FUNCTION_BLOCK FB_ErrorList

VAR_INPUT
	En : BOOL;											//Enable input
	bReset : BOOL;										//Delete all Error entry
	lErrorID : ULINT;									//ErrorID to be acknoledged
	bACK : BOOL;										//Acknoledge the given error and delete it from the list
END_VAR
	
VAR_OUTPUT
	EnO : BOOL;											//Enable output
	nNoError: UINT;										//Number of Errors
	nNoOverflow : INT;									//Number of Overflows
	pErrorSystem : POINTER TO ST_ErrorSystem;			//Pointer to ErrorSystem
END_VAR

VAR
	nFreePos : UINT;									//Number of free position in the list
	nListCnt1 : UINT;									//work variable
	ErrorSystem : ST_ErrorSystem;						//Data structure of the Error list
END_VAR

(*
* ================================================================================
*                                   DESCRIPTION
* ================================================================================
* This Function Block implements the core structure of the Error/Warning Handling
* system. It realizes the datastructure containing every Error Entry, collect
* statistics about the usage and manage the Error Entries.
* Note: The system is under development, most of the functionalities are not
* implemented or existing functionalities may change with the advance of the
* development.
* ================================================================================
*)
EnO := En;

//Ponter to ErrorSystem
pErrorSystem := ADR(ErrorSystem);

//Number of overflows
nNoOverflow := ErrorSystem.nNoOverflows;

IF bReset THEN
	MEMSET ( ADR(ErrorSystem.aErrorData[0]), 0, GVL_ErrorSystem.cSizeOfErrorData * SIZEOF(DUT_TerminalError));
	ErrorSystem.lNextErrorID := 1;
END_IF

//Number of errors in the system
nNoError := 0;
FOR nListCnt1 := 0 TO GVL_ErrorSystem.cSizeOfErrorData - 1 DO
	IF ErrorSystem.aErrorData[nListCnt1].Error_ID <> 0  THEN
		nNoError := nNoError+1; 
	END_IF
END_FOR
ErrorSystem.nNoErrors := nNoError;

//Number of free position in the list
nFreePos := GVL_ErrorSystem.cSizeOfErrorData - nNoError;

//Acknoledge specified Error entry
IF bACK THEN
	FOR nListCnt1 := 0 TO GVL_ErrorSystem.cSizeOfErrorData - 1 DO
		IF ErrorSystem.aErrorData[nListCnt1].Error_ID = lErrorID THEN
			ErrorSystem.aErrorData[nListCnt1].ErrorState := DUT_ErrorState.Acknoledged;
		END_IF
	END_FOR
END_IF

//Deleting acknoledged errors
FOR nListCnt1 := 0 TO GVL_ErrorSystem.cSizeOfErrorData - 1 DO
	IF ErrorSystem.aErrorData[nListCnt1].ErrorState = DUT_ErrorState.Acknoledged THEN
		MEMMOVE (ADR(ErrorSystem.aErrorData[nListCnt1]), ADR(ErrorSystem.aErrorData[nListCnt1+1]), (GVL_ErrorSystem.cSizeOfErrorData - 1 - nListCnt1) * SIZEOF(DUT_TerminalError));
		MEMSET(ADR(ErrorSystem.aErrorData[GVL_ErrorSystem.cSizeOfErrorData - 1]), 0, SIZEOF(DUT_TerminalError));
	END_IF
END_FOR

END_FUNCTION_BLOCK

(* stored: Version 1.1.0.1, ProductVersion 3.1.4022.6
   POU FB_ErrorList: Id {978ea49f-a940-4b4e-9f45-8cdde4adcf37}, SpecialFunc None *)
